{attribute 'GeneratedUsingTerminal: EK1100-0000-0018'}
{attribute addProperty BoxType "EK1100-0000-0018"}
{attribute addProperty Id "Beckhoff_EJx9xxEK1122Beckhoff_EJx9xxEK1122_EEA9E9F52A_0001_EJ1914_0000_0017EJ1914_0821024F34A_0002_EJ1914_0000_0018EJ1914_0821024F34A_0003_EJ1918_0000_0017EJ1918_57845E7942A_0004_EJ1918_0000_0018EJ1918_57845E7942A_0005_EJ1957_0000_0017EJ1957_9A95FC5954A_0006_EJ1957_0000_0018EJ1957_9A95FC5954A_0007_EJ2914_0000_0017EJ2914_475777A038A_0008_EJ2914_0000_0018EJ2914_475777A038A_0009_EJ2918_0000_0017EJ2918_B661C90A48A_0010_EJ2918_0000_0018EJ2918_B661C90A48A_0011_EJ6910_0000_0018EJ6910_CD4DE20014A_0012_EJ6910_0000_0020EJ6910_CD4DE20014"}
{attribute addProperty CRC "1725514541"}
{attribute addProperty Size "462"}
TYPE Beckhoff_EJx9xx_66D9432D EXTENDS EK1100_1FC0878B :
STRUCT
	{attribute addProperty Name "Beckhoff_EJx9xxEK1122"}
	Beckhoff_EJx9xxEK1122 : Beckhoff_EJx9xxEK1122_EEA9E9F5;
	{attribute addProperty Name "A_0001_EJ1914_0000_0017"}
	A_0001_EJ1914_0000_0017 : EJ1914_0821024F;
	{attribute addProperty Name "A_0002_EJ1914_0000_0018"}
	A_0002_EJ1914_0000_0018 : EJ1914_0821024F;
	{attribute addProperty Name "A_0003_EJ1918_0000_0017"}
	A_0003_EJ1918_0000_0017 : EJ1918_57845E79;
	{attribute addProperty Name "A_0004_EJ1918_0000_0018"}
	A_0004_EJ1918_0000_0018 : EJ1918_57845E79;
	{attribute addProperty Name "A_0005_EJ1957_0000_0017"}
	A_0005_EJ1957_0000_0017 : EJ1957_9A95FC59;
	{attribute addProperty Name "A_0006_EJ1957_0000_0018"}
	A_0006_EJ1957_0000_0018 : EJ1957_9A95FC59;
	{attribute addProperty Name "A_0007_EJ2914_0000_0017"}
	A_0007_EJ2914_0000_0017 : EJ2914_475777A0;
	{attribute addProperty Name "A_0008_EJ2914_0000_0018"}
	A_0008_EJ2914_0000_0018 : EJ2914_475777A0;
	{attribute addProperty Name "A_0009_EJ2918_0000_0017"}
	A_0009_EJ2918_0000_0017 : EJ2918_B661C90A;
	{attribute addProperty Name "A_0010_EJ2918_0000_0018"}
	A_0010_EJ2918_0000_0018 : EJ2918_B661C90A;
	{attribute addProperty Name "A_0011_EJ6910_0000_0018"}
	A_0011_EJ6910_0000_0018 : EJ6910_CD4DE200;
	{attribute addProperty Name "A_0012_EJ6910_0000_0020"}
	A_0012_EJ6910_0000_0020 : EJ6910_CD4DE200;
END_STRUCT
END_TYPE

(* stored: Version 1.2.0.0, ProductVersion 3.1.4024.9
   DUT Beckhoff_EJx9xx_66D9432D: Id {57b6cce8-f04b-4626-93d5-dbdb75a022a8} *)
